(* PLC project marvel_services, Institute of Astronomy Onto 0.0.1 *)
(* stored: creationDateTime 2025-01-01T00:00:00.0, modificationDateTime 2025-01-01T00:00:00.0 *)

{attribute 'qualified_only'}
TYPE ServicesMeteoSimulation : (PHOTOMETRIC := 0, DRY_WINDY := 1, DRY_TOO_WINDY := 2, WET_WINDY := 3) BYTE;
END_TYPE

TYPE ServicesParts : STRUCT
  {attribute 'TcHmiSymbol.Show'}
  timing : ServicesTiming;  (* Timing service *)
  {attribute 'TcHmiSymbol.Show'}
  mercatorMeteo : ServicesMercatorMeteo;  (* Mercator meteo service *)
  {attribute 'TcHmiSymbol.Show'}
  configManager : ConfigManager;  (* The config manager (to load/save/activate configuration data) *)
END_STRUCT;
END_TYPE

TYPE ServicesProcesses : STRUCT
  {attribute 'TcHmiSymbol.Show'}
  initialize : Process;  (* Start initializing *)
  {attribute 'TcHmiSymbol.Show'}
  lock : Process;  (* Lock the system *)
  {attribute 'TcHmiSymbol.Show'}
  unlock : Process;  (* Unlock the system *)
  {attribute 'TcHmiSymbol.Show'}
  changeOperatingState : ChangeOperatingStateProcess;  (* Change the operating state (e.g. AUTO, MANUAL, ...) *)
END_STRUCT;
END_TYPE

TYPE ServicesTimingProcesses : STRUCT

END_STRUCT;
END_TYPE

TYPE ServicesMercatorMeteoProcesses : STRUCT

END_STRUCT;
END_TYPE

TYPE ServicesStatuses : STRUCT
  {attribute 'OPC.UA.DA' := '1'}
  {attribute 'OPC.UA.DA.Access' := '1'}
  {attribute 'TcHmiSymbol.Show'}
  init : InitializationStatus;
  {attribute 'OPC.UA.DA' := '1'}
  {attribute 'OPC.UA.DA.Access' := '1'}
  {attribute 'TcHmiSymbol.Show'}
  health : HealthStatus;
  {attribute 'OPC.UA.DA' := '1'}
  {attribute 'OPC.UA.DA.Access' := '1'}
  {attribute 'TcHmiSymbol.Show'}
  busy : BusyStatus;
  {attribute 'OPC.UA.DA' := '1'}
  {attribute 'OPC.UA.DA.Access' := '1'}
  {attribute 'TcHmiSymbol.Show'}
  operating : OperatingStatus;
END_STRUCT;
END_TYPE

TYPE ServicesTimingStatuses : STRUCT
  {attribute 'OPC.UA.DA' := '1'}
  {attribute 'OPC.UA.DA.Access' := '1'}
  {attribute 'TcHmiSymbol.Show'}
  health : HealthStatus;
END_STRUCT;
END_TYPE

TYPE ServicesMercatorMeteoMeasurementStatuses : STRUCT
  {attribute 'OPC.UA.DA' := '1'}
  {attribute 'OPC.UA.DA.Access' := '1'}
  {attribute 'TcHmiSymbol.Show'}
  enabled : EnabledStatus;  (* Is the temperature being measured? *)
  {attribute 'OPC.UA.DA' := '1'}
  {attribute 'OPC.UA.DA.Access' := '1'}
  {attribute 'TcHmiSymbol.Show'}
  health : HealthStatus;  (* Is the data valid and within range? *)
  {attribute 'OPC.UA.DA' := '1'}
  {attribute 'OPC.UA.DA.Access' := '1'}
  {attribute 'TcHmiSymbol.Show'}
  alarm : HiHiLoLoAlarmStatus;  (* Alarm status *)
END_STRUCT;
END_TYPE

TYPE ServicesMercatorMeteoStatuses : STRUCT
  {attribute 'OPC.UA.DA' := '1'}
  {attribute 'OPC.UA.DA.Access' := '1'}
  {attribute 'TcHmiSymbol.Show'}
  meteoHealthStatus : HealthStatus;
  {attribute 'OPC.UA.DA' := '1'}
  {attribute 'OPC.UA.DA.Access' := '1'}
  {attribute 'TcHmiSymbol.Show'}
  health : HealthStatus;
END_STRUCT;
END_TYPE

TYPE ServicesTimingConfig : STRUCT
  {attribute 'TcHmiSymbol.Show'}
  alwaysUseLocalClock : BOOL;  (* If TRUE, then the local clock (source=LOCAL_CLOCK) will be used even if an external (more accurate!) clock is available *)
END_STRUCT;
END_TYPE

TYPE ServicesMercatorMeteoConfig : STRUCT
  {attribute 'TcHmiSymbol.Show'}
  simulated : BOOL;  (* TRUE to simulate the Mercator weather station data *)
  {attribute 'TcHmiSymbol.Show'}
  enableWeatherMonitoring : BOOL;  (* Enable weather monitoring and emergency closing *)
  {attribute 'TcHmiSymbol.Show'}
  wetLimit : LREAL;  (* Wet if (rainIntensity+hailIntensity)>wetLimit *)
  {attribute 'TcHmiSymbol.Show'}
  windSpeedMinimum : MeasurementConfig;  (* Config for the wind speed minimum *)
  {attribute 'TcHmiSymbol.Show'}
  windSpeedAverage : MeasurementConfig;  (* Config for the wind speed average *)
  {attribute 'TcHmiSymbol.Show'}
  windSpeedMaximum : MeasurementConfig;  (* Config for the wind speed maximum *)
  {attribute 'TcHmiSymbol.Show'}
  windDirectionMinimum : MeasurementConfig;  (* Config for the wind direction minimum *)
  {attribute 'TcHmiSymbol.Show'}
  windDirectionAverage : MeasurementConfig;  (* Config for the wind direction average *)
  {attribute 'TcHmiSymbol.Show'}
  windDirectionMaximum : MeasurementConfig;  (* Config for the wind direction maximum *)
  {attribute 'TcHmiSymbol.Show'}
  airPressure : MeasurementConfig;  (* Config for the air pressure *)
  {attribute 'TcHmiSymbol.Show'}
  airTemperature : MeasurementConfig;  (* Config for the air temperature *)
  {attribute 'TcHmiSymbol.Show'}
  internalTemperature : MeasurementConfig;  (* Config for the internal temperature *)
  {attribute 'TcHmiSymbol.Show'}
  relativeHumidity : MeasurementConfig;  (* Config for the relative humidity *)
  {attribute 'TcHmiSymbol.Show'}
  rainAccumulation : MeasurementConfig;  (* Config for the rain accumulation *)
  {attribute 'TcHmiSymbol.Show'}
  rainDuration : MeasurementConfig;  (* Config for the rain duration *)
  {attribute 'TcHmiSymbol.Show'}
  rainIntensity : MeasurementConfig;  (* Config for the rain intensity *)
  {attribute 'TcHmiSymbol.Show'}
  rainPeakIntensity : MeasurementConfig;  (* Config for the rain peak intensity *)
  {attribute 'TcHmiSymbol.Show'}
  hailAccumulation : MeasurementConfig;  (* Config for the hail accumulation *)
  {attribute 'TcHmiSymbol.Show'}
  hailDuration : MeasurementConfig;  (* Config for the hail duration *)
  {attribute 'TcHmiSymbol.Show'}
  hailIntensity : MeasurementConfig;  (* Config for the hail intensity *)
  {attribute 'TcHmiSymbol.Show'}
  hailPeakIntensity : MeasurementConfig;  (* Config for the hail peak intensity *)
  {attribute 'TcHmiSymbol.Show'}
  heatingTemperature : MeasurementConfig;  (* Config for the heating temperature *)
  {attribute 'TcHmiSymbol.Show'}
  heatingVoltage : MeasurementConfig;  (* Config for the heating voltage *)
  {attribute 'TcHmiSymbol.Show'}
  supplyVoltage : MeasurementConfig;  (* Config for the supply voltage *)
  {attribute 'TcHmiSymbol.Show'}
  referenceVoltage : MeasurementConfig;  (* Config for the 3.5 V reference voltage *)
  {attribute 'TcHmiSymbol.Show'}
  dewpoint : MeasurementConfig;  (* Config for the dew point *)
END_STRUCT;
END_TYPE

TYPE ServicesConfig : STRUCT
  {attribute 'TcHmiSymbol.Show'}
  timing : ServicesTimingConfig;  (* Timing config *)
  {attribute 'TcHmiSymbol.Show'}
  mercatorMeteo : ServicesMercatorMeteoConfig;  (* Mercator meteo config *)
END_STRUCT;
END_TYPE

FUNCTION_BLOCK SM_Services
  VAR_INPUT
    {attribute 'TcHmiSymbol.Show'}
    {attribute 'OPC.UA.DA' := '1'}
    {attribute 'OPC.UA.DA.Access' := '1'}
    editableConfig : ServicesConfig;  (* Editable configuration of the Services subsystem *)
  END_VAR
  VAR_OUTPUT
    {attribute 'OPC.UA.DA' := '1'}
    {attribute 'OPC.UA.DA.Access' := '1'}
    {attribute 'TcHmiSymbol.Show'}
    actualStatus : STRING;  (* Current status description *)
    {attribute 'TcHmiSymbol.Hide'}
    {attribute 'OPC.UA.DA' := '0'}
    previousStatus : STRING;  (* Previous status description *)
    {attribute 'TcHmiSymbol.Show'}
    {attribute 'OPC.UA.DA' := '1'}
    {attribute 'OPC.UA.DA.Access' := '1'}
    config : ServicesConfig;  (* Active configuration of the Services subsystem *)
    {attribute 'TcHmiSymbol.Show'}
    stat : ServicesStatuses;  (* Statuses of the state machine *)
    {attribute 'TcHmiSymbol.Show'}
    parts : ServicesParts;  (* Parts of the state machine *)
    {attribute 'TcHmiSymbol.Show'}
    proc : ServicesProcesses;  (* Processes of the state machine *)
  END_VAR
  VAR_IN_OUT
    {attribute 'TcHmiSymbol.Show'}
    {attribute 'OPC.UA.DA' := '0'}
    {attribute 'TcHmiSymbol.Hide'}
    operator_ref : OperatorStatus;  (* Shared operator status *)
  END_VAR

            parts.timing(
    operator_ref := operator_ref,
    config_ref := config.timing);
parts.mercatorMeteo( config_ref := config.mercatorMeteo );
parts.configManager( isEnabled := operator_ref = OperatorStatus.tech );
stat.health := F_HealthStatus(
    superState := TRUE,
    isGood := (parts.timing.stat.health = HealthStatus.good) AND (parts.mercatorMeteo.stat.health = HealthStatus.good),
    hasWarning := (parts.timing.stat.health = HealthStatus.warning) OR (parts.mercatorMeteo.stat.health = HealthStatus.warning));
stat.busy := F_BusyStatus(
    superState := TRUE,
    isBusy := stat.init = InitializationStatus.initializing);
proc.initialize( isEnabled := (stat.init = InitializationStatus.shutdown) OR ((stat.init = InitializationStatus.initializingFailed) OR (stat.init = InitializationStatus.initialized)) );
proc.lock( isEnabled := (operator_ref = OperatorStatus.tech) AND (stat.init = InitializationStatus.initialized) );
proc.unlock( isEnabled := (operator_ref = OperatorStatus.tech) AND (stat.init = InitializationStatus.locked) );
proc.changeOperatingState( isEnabled := FALSE );

          
END_FUNCTION_BLOCK

FUNCTION_BLOCK SM_ServicesTiming
  VAR_INPUT
    {attribute 'TcHmiSymbol.Show'}
    {attribute 'OPC.UA.DA' := '1'}
    {attribute 'OPC.UA.DA.Access' := '1'}
    ntpExtTime AT %I* : LINT;  (* TcCOM object nExtTime variable *)
    {attribute 'TcHmiSymbol.Show'}
    {attribute 'OPC.UA.DA' := '1'}
    {attribute 'OPC.UA.DA.Access' := '1'}
    isNtpConnected AT %I* : BOOL;  (* TRUE if NTP is connected *)
    {attribute 'TcHmiSymbol.Show'}
    {attribute 'OPC.UA.DA' := '1'}
    {attribute 'OPC.UA.DA.Access' := '1'}
    isNtpSynchronized AT %I* : BOOL;  (* TRUE if NTP is synchronized *)
  END_VAR
  VAR_OUTPUT
    {attribute 'OPC.UA.DA' := '1'}
    {attribute 'OPC.UA.DA.Access' := '1'}
    {attribute 'TcHmiSymbol.Show'}
    actualStatus : STRING;  (* Current status description *)
    {attribute 'TcHmiSymbol.Hide'}
    {attribute 'OPC.UA.DA' := '0'}
    previousStatus : STRING;  (* Previous status description *)
    {attribute 'TcHmiSymbol.Show'}
    {attribute 'OPC.UA.DA' := '1'}
    {attribute 'OPC.UA.DA.Access' := '1'}
    utcDateString : STRING;  (* UTC date as a string of format YYYY-MM-DD *)
    {attribute 'TcHmiSymbol.Show'}
    {attribute 'OPC.UA.DA' := '1'}
    {attribute 'OPC.UA.DA.Access' := '1'}
    utcTimeString : STRING;  (* UTC time as a string of format HH-MM-SS.SSS *)
    {attribute 'TcHmiSymbol.Show'}
    stat : ServicesTimingStatuses;  (* Statuses of the state machine *)
    {attribute 'TcHmiSymbol.Show'}
    proc : ServicesTimingProcesses;  (* Processes of the state machine *)
  END_VAR
  VAR_IN_OUT
    {attribute 'TcHmiSymbol.Show'}
    {attribute 'OPC.UA.DA' := '0'}
    {attribute 'TcHmiSymbol.Hide'}
    operator_ref : OperatorStatus;  (* Shared operator status *)
    {attribute 'TcHmiSymbol.Show'}
    {attribute 'OPC.UA.DA' := '0'}
    {attribute 'TcHmiSymbol.Hide'}
    config_ref : ServicesTimingConfig;  (* The config *)
  END_VAR
  VAR
    {attribute 'TcHmiSymbol.Show'}
    {attribute 'OPC.UA.DA' := '1'}
    {attribute 'OPC.UA.DA.Access' := '1'}
    ntpExtTime_ro : LINT;
    {attribute 'TcHmiSymbol.Show'}
    {attribute 'OPC.UA.DA' := '1'}
    {attribute 'OPC.UA.DA.Access' := '1'}
    isNtpConnected_ro : BOOL;
    {attribute 'TcHmiSymbol.Show'}
    {attribute 'OPC.UA.DA' := '1'}
    {attribute 'OPC.UA.DA.Access' := '1'}
    isNtpSynchronized_ro : BOOL;
  END_VAR

            stat.health := F_HealthStatus(
    superState := TRUE,
    hasWarning := FALSE,
    isGood := isNtpConnected AND isNtpSynchronized);
ntpExtTime_ro := ntpExtTime;
isNtpConnected_ro := isNtpConnected;
isNtpSynchronized_ro := isNtpSynchronized;

          
END_FUNCTION_BLOCK

FUNCTION_BLOCK SM_ServicesMercatorMeteoMeasurement
  VAR_INPUT
    {attribute 'TcHmiSymbol.Show'}
    {attribute 'OPC.UA.DA' := '1'}
    {attribute 'OPC.UA.DA.Access' := '1'}
    data : LREAL;  (* The measured data *)
    {attribute 'TcHmiSymbol.Show'}
    {attribute 'OPC.UA.DA' := '1'}
    {attribute 'OPC.UA.DA.Access' := '1'}
    valid : BOOL;  (* TRUE if the data is valid *)
    {attribute 'TcHmiSymbol.Show'}
    {attribute 'OPC.UA.DA' := '1'}
    {attribute 'OPC.UA.DA.Access' := '1'}
    disconnected : BOOL;  (* TRUE if the data provider is disconnected *)
  END_VAR
  VAR_OUTPUT
    {attribute 'OPC.UA.DA' := '1'}
    {attribute 'OPC.UA.DA.Access' := '1'}
    {attribute 'TcHmiSymbol.Show'}
    actualStatus : STRING;  (* Current status description *)
    {attribute 'TcHmiSymbol.Hide'}
    {attribute 'OPC.UA.DA' := '0'}
    previousStatus : STRING;  (* Previous status description *)
    {attribute 'TcHmiSymbol.Show'}
    stat : ServicesMercatorMeteoMeasurementStatuses;  (* Statuses of the state machine *)
  END_VAR
  VAR_IN_OUT
    {attribute 'TcHmiSymbol.Show'}
    {attribute 'OPC.UA.DA' := '0'}
    {attribute 'TcHmiSymbol.Hide'}
    config_ref : MeasurementConfig;  (* Reference to the config *)
  END_VAR

            stat.enabled := F_EnabledStatus(
    superState := TRUE,
    isEnabled := config_ref.enabled);
stat.health := F_HealthStatus(
    superState := stat.enabled = EnabledStatus.enabled,
    isGood := NOT((NOT(valid)) OR (disconnected OR ((stat.alarm = HiHiLoLoAlarmStatus.hiHi) OR (stat.alarm = HiHiLoLoAlarmStatus.loLo)))),
    hasWarning := (stat.alarm = HiHiLoLoAlarmStatus.hi) OR (stat.alarm = HiHiLoLoAlarmStatus.lo));
stat.alarm := F_HiHiLoLoAlarmStatus(
    superState := stat.enabled = EnabledStatus.enabled,
    config := config_ref.alarms,
    value := data);

          
END_FUNCTION_BLOCK

FUNCTION_BLOCK SM_ServicesMercatorMeteo
  VAR_INPUT
    {attribute 'TcHmiSymbol.Show'}
    {attribute 'OPC.UA.DA' := '1'}
    {attribute 'OPC.UA.DA.Access' := '1'}
    weatherStatus : STRING;  (* Weather status as a string *)
    {attribute 'TcHmiSymbol.Show'}
    {attribute 'OPC.UA.DA' := '1'}
    {attribute 'OPC.UA.DA.Access' := '1'}
    mercatorConnected : BOOL;  (* True if MTCS is connected *)
    {attribute 'TcHmiSymbol.Show'}
    {attribute 'OPC.UA.DA' := '1'}
    {attribute 'OPC.UA.DA.Access' := '1'}
    windSpeedMinimum : ServicesMercatorMeteoMeasurement;  (* Wind speed minimum *)
    {attribute 'TcHmiSymbol.Show'}
    {attribute 'OPC.UA.DA' := '1'}
    {attribute 'OPC.UA.DA.Access' := '1'}
    windSpeedAverage : ServicesMercatorMeteoMeasurement;  (* Wind speed average *)
    {attribute 'TcHmiSymbol.Show'}
    {attribute 'OPC.UA.DA' := '1'}
    {attribute 'OPC.UA.DA.Access' := '1'}
    windSpeedMaximum : ServicesMercatorMeteoMeasurement;  (* Wind speed maximum *)
    {attribute 'TcHmiSymbol.Show'}
    {attribute 'OPC.UA.DA' := '1'}
    {attribute 'OPC.UA.DA.Access' := '1'}
    windDirectionMinimum : ServicesMercatorMeteoMeasurement;  (* Wind direction minimum *)
    {attribute 'TcHmiSymbol.Show'}
    {attribute 'OPC.UA.DA' := '1'}
    {attribute 'OPC.UA.DA.Access' := '1'}
    windDirectionAverage : ServicesMercatorMeteoMeasurement;  (* Wind direction average *)
    {attribute 'TcHmiSymbol.Show'}
    {attribute 'OPC.UA.DA' := '1'}
    {attribute 'OPC.UA.DA.Access' := '1'}
    windDirectionMaximum : ServicesMercatorMeteoMeasurement;  (* Wind direction maximum *)
    {attribute 'TcHmiSymbol.Show'}
    {attribute 'OPC.UA.DA' := '1'}
    {attribute 'OPC.UA.DA.Access' := '1'}
    airPressure : ServicesMercatorMeteoMeasurement;  (* Air pressure *)
    {attribute 'TcHmiSymbol.Show'}
    {attribute 'OPC.UA.DA' := '1'}
    {attribute 'OPC.UA.DA.Access' := '1'}
    airTemperature : ServicesMercatorMeteoMeasurement;  (* Air temperature *)
    {attribute 'TcHmiSymbol.Show'}
    {attribute 'OPC.UA.DA' := '1'}
    {attribute 'OPC.UA.DA.Access' := '1'}
    internalTemperature : ServicesMercatorMeteoMeasurement;  (* Internal temperature *)
    {attribute 'TcHmiSymbol.Show'}
    {attribute 'OPC.UA.DA' := '1'}
    {attribute 'OPC.UA.DA.Access' := '1'}
    relativeHumidity : ServicesMercatorMeteoMeasurement;  (* Relative humidity *)
    {attribute 'TcHmiSymbol.Show'}
    {attribute 'OPC.UA.DA' := '1'}
    {attribute 'OPC.UA.DA.Access' := '1'}
    rainAccumulation : ServicesMercatorMeteoMeasurement;  (* Rain accumulation *)
    {attribute 'TcHmiSymbol.Show'}
    {attribute 'OPC.UA.DA' := '1'}
    {attribute 'OPC.UA.DA.Access' := '1'}
    rainDuration : ServicesMercatorMeteoMeasurement;  (* Rain duration *)
    {attribute 'TcHmiSymbol.Show'}
    {attribute 'OPC.UA.DA' := '1'}
    {attribute 'OPC.UA.DA.Access' := '1'}
    rainIntensity : ServicesMercatorMeteoMeasurement;  (* Rain intensity *)
    {attribute 'TcHmiSymbol.Show'}
    {attribute 'OPC.UA.DA' := '1'}
    {attribute 'OPC.UA.DA.Access' := '1'}
    rainPeakIntensity : ServicesMercatorMeteoMeasurement;  (* Rain peak intensity *)
    {attribute 'TcHmiSymbol.Show'}
    {attribute 'OPC.UA.DA' := '1'}
    {attribute 'OPC.UA.DA.Access' := '1'}
    hailAccumulation : ServicesMercatorMeteoMeasurement;  (* Hail accumulation *)
    {attribute 'TcHmiSymbol.Show'}
    {attribute 'OPC.UA.DA' := '1'}
    {attribute 'OPC.UA.DA.Access' := '1'}
    hailDuration : ServicesMercatorMeteoMeasurement;  (* Hail duration *)
    {attribute 'TcHmiSymbol.Show'}
    {attribute 'OPC.UA.DA' := '1'}
    {attribute 'OPC.UA.DA.Access' := '1'}
    hailIntensity : ServicesMercatorMeteoMeasurement;  (* Hail intensity *)
    {attribute 'TcHmiSymbol.Show'}
    {attribute 'OPC.UA.DA' := '1'}
    {attribute 'OPC.UA.DA.Access' := '1'}
    hailPeakIntensity : ServicesMercatorMeteoMeasurement;  (* Hail peak intensity *)
    {attribute 'TcHmiSymbol.Show'}
    {attribute 'OPC.UA.DA' := '1'}
    {attribute 'OPC.UA.DA.Access' := '1'}
    heatingTemperature : ServicesMercatorMeteoMeasurement;  (* Heating temperature *)
    {attribute 'TcHmiSymbol.Show'}
    {attribute 'OPC.UA.DA' := '1'}
    {attribute 'OPC.UA.DA.Access' := '1'}
    heatingVoltage : ServicesMercatorMeteoMeasurement;  (* Heating voltage *)
    {attribute 'TcHmiSymbol.Show'}
    {attribute 'OPC.UA.DA' := '1'}
    {attribute 'OPC.UA.DA.Access' := '1'}
    supplyVoltage : ServicesMercatorMeteoMeasurement;  (* Supply voltage *)
    {attribute 'TcHmiSymbol.Show'}
    {attribute 'OPC.UA.DA' := '1'}
    {attribute 'OPC.UA.DA.Access' := '1'}
    referenceVoltage : ServicesMercatorMeteoMeasurement;  (* Reference voltage *)
    {attribute 'TcHmiSymbol.Show'}
    {attribute 'OPC.UA.DA' := '1'}
    {attribute 'OPC.UA.DA.Access' := '1'}
    dewpoint : ServicesMercatorMeteoMeasurement;  (* Calculated dew point temperature *)
    {attribute 'TcHmiSymbol.Show'}
    {attribute 'OPC.UA.DA' := '1'}
    {attribute 'OPC.UA.DA.Access' := '1'}
    durationOK : Duration;  (* Duration that the meteo is OK *)
    {attribute 'TcHmiSymbol.Show'}
    {attribute 'OPC.UA.DA' := '1'}
    {attribute 'OPC.UA.DA.Access' := '1'}
    wet : BOOL;  (* Wet if (rainIntensity+hailIntensity) > config.wetLimit *)
    {attribute 'TcHmiSymbol.Show'}
    {attribute 'OPC.UA.DA' := '1'}
    {attribute 'OPC.UA.DA.Access' := '1'}
    heating : BOOL;  (* Heating or not? *)
    {attribute 'TcHmiSymbol.Show'}
    {attribute 'OPC.UA.DA' := '1'}
    {attribute 'OPC.UA.DA.Access' := '1'}
    windDirectionMinimumString : STRING;  (* Average direction of the wind as a string *)
    {attribute 'TcHmiSymbol.Show'}
    {attribute 'OPC.UA.DA' := '1'}
    {attribute 'OPC.UA.DA.Access' := '1'}
    windDirectionAverageString : STRING;  (* Average direction of the wind as a string *)
    {attribute 'TcHmiSymbol.Show'}
    {attribute 'OPC.UA.DA' := '1'}
    {attribute 'OPC.UA.DA.Access' := '1'}
    windDirectionMaximumString : STRING;  (* Average direction of the wind as a string *)
    {attribute 'TcHmiSymbol.Show'}
    {attribute 'OPC.UA.DA' := '1'}
    {attribute 'OPC.UA.DA.Access' := '1'}
    fromSimulation : MercatorMeteoExchange;  (* The simulated data (if config.simulated is TRUE) *)
    {attribute 'OPC.UA.DA' := '0'}
    {attribute 'TcHmiSymbol.Hide'}
    fromMercator AT %I* : MercatorMeteoExchange;  (* The data exchanged by the Mercator telescope *)
    {attribute 'OPC.UA.DA' := '0'}
    {attribute 'TcHmiSymbol.Hide'}
    mercatorDisconnected AT %I* : BOOL;  (* The data exchanged by the Mercator telescope is invalid *)
  END_VAR
  VAR_OUTPUT
    {attribute 'OPC.UA.DA' := '1'}
    {attribute 'OPC.UA.DA.Access' := '1'}
    {attribute 'TcHmiSymbol.Show'}
    actualStatus : STRING;  (* Current status description *)
    {attribute 'TcHmiSymbol.Hide'}
    {attribute 'OPC.UA.DA' := '0'}
    previousStatus : STRING;  (* Previous status description *)
    {attribute 'TcHmiSymbol.Show'}
    stat : ServicesMercatorMeteoStatuses;  (* Statuses of the state machine *)
    {attribute 'TcHmiSymbol.Show'}
    proc : ServicesMercatorMeteoProcesses;  (* Processes of the state machine *)
  END_VAR
  VAR_IN_OUT
    {attribute 'TcHmiSymbol.Show'}
    {attribute 'OPC.UA.DA' := '0'}
    {attribute 'TcHmiSymbol.Hide'}
    config_ref : ServicesMercatorMeteoConfig;  (* The config *)
  END_VAR
  VAR
    {attribute 'OPC.UA.DA' := '0'}
    {attribute 'TcHmiSymbol.Hide'}
    fromMercator_ro : MercatorMeteoExchange;
    {attribute 'OPC.UA.DA' := '0'}
    {attribute 'TcHmiSymbol.Hide'}
    mercatorDisconnected_ro : BOOL;
  END_VAR

            windSpeedMinimum(
    config_ref := config_ref.windSpeedMinimum,
    data := fromMercator.windSpeedMinimum,
    valid := fromMercator.windSpeedMinimumValid,
    disconnected := mercatorDisconnected);
windSpeedAverage(
    config_ref := config_ref.windSpeedAverage,
    data := fromMercator.windSpeedAverage,
    valid := fromMercator.windSpeedAverageValid,
    disconnected := mercatorDisconnected);
windSpeedMaximum(
    config_ref := config_ref.windSpeedMaximum,
    data := fromMercator.windSpeedMaximum,
    valid := fromMercator.windSpeedMaximumValid,
    disconnected := mercatorDisconnected);
windDirectionMinimum(
    config_ref := config_ref.windDirectionMinimum,
    data := fromMercator.windDirectionMinimum,
    valid := fromMercator.windDirectionMinimumValid,
    disconnected := mercatorDisconnected);
windDirectionAverage(
    config_ref := config_ref.windDirectionAverage,
    data := fromMercator.windDirectionAverage,
    valid := fromMercator.windDirectionAverageValid,
    disconnected := mercatorDisconnected);
windDirectionMaximum(
    config_ref := config_ref.windDirectionMaximum,
    data := fromMercator.windDirectionMaximum,
    valid := fromMercator.windDirectionMaximumValid,
    disconnected := mercatorDisconnected);
airPressure(
    config_ref := config_ref.airPressure,
    data := fromMercator.airPressure,
    valid := fromMercator.airPressureValid,
    disconnected := mercatorDisconnected);
airTemperature(
    config_ref := config_ref.airTemperature,
    data := fromMercator.airTemperature,
    valid := fromMercator.airTemperatureValid,
    disconnected := mercatorDisconnected);
internalTemperature(
    config_ref := config_ref.internalTemperature,
    data := fromMercator.internalTemperature,
    valid := fromMercator.internalTemperatureValid,
    disconnected := mercatorDisconnected);
relativeHumidity(
    config_ref := config_ref.relativeHumidity,
    data := fromMercator.relativeHumidity,
    valid := fromMercator.relativeHumidityValid,
    disconnected := mercatorDisconnected);
rainAccumulation(
    config_ref := config_ref.rainAccumulation,
    data := fromMercator.rainAccumulation,
    valid := fromMercator.rainAccumulationValid,
    disconnected := mercatorDisconnected);
rainDuration(
    config_ref := config_ref.rainDuration,
    data := fromMercator.rainDuration,
    valid := fromMercator.rainDurationValid,
    disconnected := mercatorDisconnected);
rainIntensity(
    config_ref := config_ref.rainIntensity,
    data := fromMercator.rainIntensity,
    valid := fromMercator.rainIntensityValid,
    disconnected := mercatorDisconnected);
rainPeakIntensity(
    config_ref := config_ref.rainPeakIntensity,
    data := fromMercator.rainPeakIntensity,
    valid := fromMercator.rainPeakIntensityValid,
    disconnected := mercatorDisconnected);
hailAccumulation(
    config_ref := config_ref.hailAccumulation,
    data := fromMercator.hailAccumulation,
    valid := fromMercator.hailAccumulationValid,
    disconnected := mercatorDisconnected);
hailDuration(
    config_ref := config_ref.hailDuration,
    data := fromMercator.hailDuration,
    valid := fromMercator.hailDurationValid,
    disconnected := mercatorDisconnected);
hailIntensity(
    config_ref := config_ref.hailIntensity,
    data := fromMercator.hailIntensity,
    valid := fromMercator.hailIntensityValid,
    disconnected := mercatorDisconnected);
hailPeakIntensity(
    config_ref := config_ref.hailPeakIntensity,
    data := fromMercator.hailPeakIntensity,
    valid := fromMercator.hailPeakIntensityValid,
    disconnected := mercatorDisconnected);
heatingTemperature(
    config_ref := config_ref.heatingTemperature,
    data := fromMercator.heatingTemperature,
    valid := fromMercator.heatingTemperatureValid,
    disconnected := mercatorDisconnected);
heatingVoltage(
    config_ref := config_ref.heatingVoltage,
    data := fromMercator.heatingVoltage,
    valid := fromMercator.heatingVoltageValid,
    disconnected := mercatorDisconnected);
supplyVoltage(
    config_ref := config_ref.supplyVoltage,
    data := fromMercator.supplyVoltage,
    valid := fromMercator.supplyVoltageValid,
    disconnected := mercatorDisconnected);
referenceVoltage(
    config_ref := config_ref.referenceVoltage,
    data := fromMercator.referenceVoltage,
    valid := fromMercator.referenceVoltageValid,
    disconnected := mercatorDisconnected);
dewpoint(
    config_ref := config_ref.dewpoint,
    data := fromMercator.dewpoint,
    valid := fromMercator.dewpointValid,
    disconnected := mercatorDisconnected);
stat.meteoHealthStatus := F_HealthStatus(
    superState := stat.health = HealthStatus.good,
    isGood := ((windSpeedMinimum.stat.health = HealthStatus.good) OR (windSpeedMinimum.stat.enabled = EnabledStatus.disabled)) AND (((windSpeedAverage.stat.health = HealthStatus.good) OR (windSpeedAverage.stat.enabled = EnabledStatus.disabled)) AND (((windSpeedMaximum.stat.health = HealthStatus.good) OR (windSpeedMaximum.stat.enabled = EnabledStatus.disabled)) AND (((windDirectionMinimum.stat.health = HealthStatus.good) OR (windDirectionMinimum.stat.enabled = EnabledStatus.disabled)) AND (((windDirectionAverage.stat.health = HealthStatus.good) OR (windDirectionAverage.stat.enabled = EnabledStatus.disabled)) AND (((windDirectionMaximum.stat.health = HealthStatus.good) OR (windDirectionMaximum.stat.enabled = EnabledStatus.disabled)) AND (((airPressure.stat.health = HealthStatus.good) OR (airPressure.stat.enabled = EnabledStatus.disabled)) AND (((airTemperature.stat.health = HealthStatus.good) OR (airTemperature.stat.enabled = EnabledStatus.disabled)) AND (((internalTemperature.stat.health = HealthStatus.good) OR (internalTemperature.stat.enabled = EnabledStatus.disabled)) AND (((relativeHumidity.stat.health = HealthStatus.good) OR (relativeHumidity.stat.enabled = EnabledStatus.disabled)) AND (((rainAccumulation.stat.health = HealthStatus.good) OR (rainAccumulation.stat.enabled = EnabledStatus.disabled)) AND (((rainDuration.stat.health = HealthStatus.good) OR (rainDuration.stat.enabled = EnabledStatus.disabled)) AND (((rainIntensity.stat.health = HealthStatus.good) OR (rainIntensity.stat.enabled = EnabledStatus.disabled)) AND (((rainPeakIntensity.stat.health = HealthStatus.good) OR (rainPeakIntensity.stat.enabled = EnabledStatus.disabled)) AND (((hailAccumulation.stat.health = HealthStatus.good) OR (hailAccumulation.stat.enabled = EnabledStatus.disabled)) AND (((hailDuration.stat.health = HealthStatus.good) OR (hailDuration.stat.enabled = EnabledStatus.disabled)) AND (((hailIntensity.stat.health = HealthStatus.good) OR (hailIntensity.stat.enabled = EnabledStatus.disabled)) AND (((hailPeakIntensity.stat.health = HealthStatus.good) OR (hailPeakIntensity.stat.enabled = EnabledStatus.disabled)) AND (((heatingTemperature.stat.health = HealthStatus.good) OR (heatingTemperature.stat.enabled = EnabledStatus.disabled)) AND (((heatingVoltage.stat.health = HealthStatus.good) OR (heatingVoltage.stat.enabled = EnabledStatus.disabled)) AND (((supplyVoltage.stat.health = HealthStatus.good) OR (supplyVoltage.stat.enabled = EnabledStatus.disabled)) AND (((referenceVoltage.stat.health = HealthStatus.good) OR (referenceVoltage.stat.enabled = EnabledStatus.disabled)) AND ((dewpoint.stat.health = HealthStatus.good) OR (dewpoint.stat.enabled = EnabledStatus.disabled))))))))))))))))))))))),
    hasWarning := (windSpeedMinimum.stat.health = HealthStatus.warning) OR ((windSpeedAverage.stat.health = HealthStatus.warning) OR ((windSpeedMaximum.stat.health = HealthStatus.warning) OR ((windDirectionMinimum.stat.health = HealthStatus.warning) OR ((windDirectionAverage.stat.health = HealthStatus.warning) OR ((windDirectionMaximum.stat.health = HealthStatus.warning) OR ((airPressure.stat.health = HealthStatus.warning) OR ((airTemperature.stat.health = HealthStatus.warning) OR ((internalTemperature.stat.health = HealthStatus.warning) OR ((relativeHumidity.stat.health = HealthStatus.warning) OR ((rainAccumulation.stat.health = HealthStatus.warning) OR ((rainDuration.stat.health = HealthStatus.warning) OR ((rainIntensity.stat.health = HealthStatus.warning) OR ((rainPeakIntensity.stat.health = HealthStatus.warning) OR ((hailAccumulation.stat.health = HealthStatus.warning) OR ((hailDuration.stat.health = HealthStatus.warning) OR ((hailIntensity.stat.health = HealthStatus.warning) OR ((hailPeakIntensity.stat.health = HealthStatus.warning) OR ((heatingTemperature.stat.health = HealthStatus.warning) OR ((heatingVoltage.stat.health = HealthStatus.warning) OR ((supplyVoltage.stat.health = HealthStatus.warning) OR ((referenceVoltage.stat.health = HealthStatus.warning) OR (dewpoint.stat.health = HealthStatus.warning)))))))))))))))))))))));
stat.health := F_HealthStatus(
    superState := TRUE,
    hasWarning := FALSE,
    isGood := fromMercator.mercatorServiceHealthy AND (NOT(mercatorDisconnected)));
fromMercator_ro := fromMercator;
mercatorDisconnected_ro := mercatorDisconnected;

          
END_FUNCTION_BLOCK
